(* PLC project SimpleCfUnitExample.project, CODESYS CODESYS V3.5 SP16 Patch 4 *)
(* stored: creationDateTime 2021-04-23T10:44:36.3809595, modificationDateTime 2021-04-23T10:43:53.8206191 *)

{attribute 'call_after_init'}
FUNCTION_BLOCK FB_Sum_Test EXTENDS CfUnit.FB_TestSuite

            TwoPlusTwoEqualsFour();
TwoPlusOneEqualsThree();
ZeroPlusZeroEqualsZero();
          

METHOD TwoPlusTwoEqualsFour
  VAR
    Sum : FB_Sum;
    Result : UINT;
    ExpectedSum : UINT := 4;
  END_VAR
                  TEST('TwoPlusTwoEqualsFour');

Sum(one := 2, two := 2, result => Result);

AssertEquals(Expected := ExpectedSum,
             Actual := Result,
             Message := 'The calculation is not correct');

TEST_FINISHED();
                
END_METHOD

METHOD TwoPlusOneEqualsThree
  VAR
    Sum : FB_Sum;
    Result : UINT;
    ExpectedSum : UINT := 3;
  END_VAR
                  TEST('TwoPlusOneEqualsThree');

Sum(one := 2, two := 1, result => Result);

AssertEquals(Expected := ExpectedSum,
             Actual := Result,
             Message := 'The calculation is not correct');

TEST_FINISHED();
                
END_METHOD

METHOD ZeroPlusZeroEqualsZero
  VAR
    Sum : FB_Sum;
    Result : UINT;
    ExpectedSum : UINT := 0;
  END_VAR
                  TEST('ZeroPlusZeroEqualsZero');

Sum(one := 0, two := 0, result => Result);

AssertEquals(Expected := ExpectedSum,
             Actual := Result,
             Message := 'The calculation is not correct');

TEST_FINISHED();
                
END_METHOD
END_FUNCTION_BLOCK
